Staubli VAL3: clkPark1.pgx

program clkPark1()
begin
  call park1()
end
